FUNCTION FLOOR2 (* This is a rounding function which returns the biggest possible integer which is less or equal to X. *)
  (* Standard: 61499-1 *)
  (* Version 1.0, 2026-09-17, Franz Höpfinger, Portiert aus OSCAT_basic FLOOR2.TcPOU - Bereichspruefung (X >= 2147483647.0 / X <= -2147483648.0) schuetzt vor DINT-Ueberlauf. *)
  PACKAGE OSCAT::Basic::POUs::Mathematical;
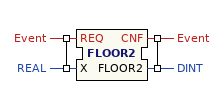
  EVENT_INPUT
    REQ WITH X;
  END_EVENT
  EVENT_OUTPUT
    CNF WITH FLOOR2;
  END_EVENT
  VAR_INPUT
    X : REAL;
  END_VAR
  VAR_OUTPUT
    FLOOR2 : DINT;
  END_VAR
  BODY IN ST:
PACKAGE OSCAT::Basic::POUs::Mathematical;

(* This is a rounding function which returns the biggest possible integer which is less or equal to X (clamped to DINT range -2147483648..2147483647). *)
FUNCTION FLOOR2 : DINT
VAR_INPUT
	X : REAL;
END_VAR

(*
 * version 1.1	4. apr. 2008 programmer 	hugo tested by		tobias
 * *
 * This is a rounding function which returns the biggest possible integer which is less or equal to X.
 * floor2(3.14) = 3 floor2(-3.14) = -4
 * Portiert 2026-09-17: Bereichspruefung schuetzt vor DINT-Ueberlauf.
 *)
IF X >= 2147483647.0 THEN
	FLOOR2 := 2147483647;
ELSIF X <= -2147483648.0 THEN
	FLOOR2 := -2147483648;
ELSE
	FLOOR2 := REAL_TO_DINT(X);
	IF DINT_TO_REAL(FLOOR2) > X THEN
		FLOOR2 := FLOOR2 - 1;
	END_IF;
END_IF;

END_FUNCTION

(* revision history hm	21. mar. 2008	rev 1.0 originlal version
 * *
 * hm	4. apr. 2008	rev 1.1 added type conversion to avoid warnings under codesys 3.0 *)
  END_BODY
END_FUNCTION
